Fanuc KAREL source: kb00003.KL

PROGRAM KB00003
%NOLOCKGROUP
VAR
P1:REAL;RESULT:REAL
BEGIN
--
P1=1.0
RESULT=ACOS(P1)
END KB00003
